Omron Sysmac Studio project NX1P2_e_NS_EmSimulação (Sysmac Studio 1.41.0.10, StandardProject)

# Controller new_Controller_0: NJ101-1020 version 1.12
Units and slaves: Power Supply : NJ-Px3001; CPU : NJ101-1020
Task PrimaryTask (priority 4, period or condition 2000): Programas

VAR_GLOBAL
    CH_Ciclo : BOOL;  (* published *)
    LMP_VM : BOOL;  (* published *)
    LMP_VD : BOOL;  (* published *)
    LMP_AM : BOOL;  (* published *)
    Chave1 : BOOL;  (* published *)
    Chave2 : BOOL;  (* published *)
    Memo_Produto1 : ARRAY[0..9] OF LREAL;  (* published *)
    Memo_Produção : ARRAY[0..9] OF LREAL;  (* published *)
    Memo_Produto2 : ARRAY[0..9] OF LREAL;  (* published *)
    TempoVM : TIME;  (* published *)
    TempoVD : TIME;  (* published *)
    TempoAM : TIME;  (* published *)
END_VAR

PROGRAM Programas
VAR
    TON_3 : TON;
    TON_1 : TON;
    TON_2 : TON;
    Ax_LMP_AM : BOOL;
END_VAR
VAR_EXTERNAL
    CH_Ciclo : BOOL;
    LMP_VM : BOOL;
    LMP_VD : BOOL;
    LMP_AM : BOOL;
    Chave1 : BOOL;
    Chave2 : BOOL;
    Memo_Produto1 : ARRAY[0..9] OF LREAL;
    Memo_Produção : ARRAY[0..9] OF LREAL;
    Memo_Produto2 : ARRAY[0..9] OF LREAL;
    TempoVM : TIME;
    TempoVD : TIME;
    TempoAM : TIME;
END_VAR
VAR
    _p1 : BOOL;
    _p2 : BOOL;
END_VAR

(* Section Semáforo: ladder, written here as Structured Text *)

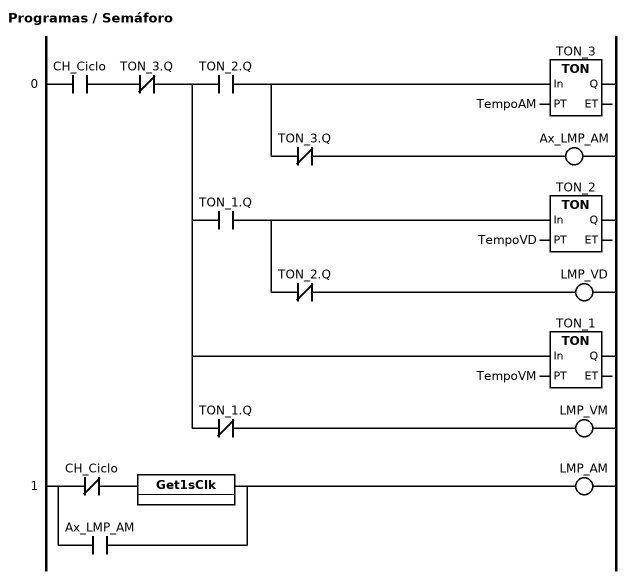
(* Rung 0 *)
_p1 := CH_Ciclo AND NOT TON_3.Q;
_p2 := CH_Ciclo AND NOT TON_3.Q AND TON_2.Q;
TON_3(In := _p2, PT := TempoAM);
Ax_LMP_AM := _p2 AND NOT TON_3.Q;
TON_2(In := _p1 AND TON_1.Q, PT := TempoVD);
LMP_VD := _p1 AND TON_1.Q AND NOT TON_2.Q;
TON_1(In := _p1, PT := TempoVM);
LMP_VM := _p1 AND NOT TON_1.Q;
(* Rung 1 *)
LMP_AM := (NOT CH_Ciclo AND Get1sClk()) OR Ax_LMP_AM;

(* Section Receita: ladder, written here as Structured Text *)

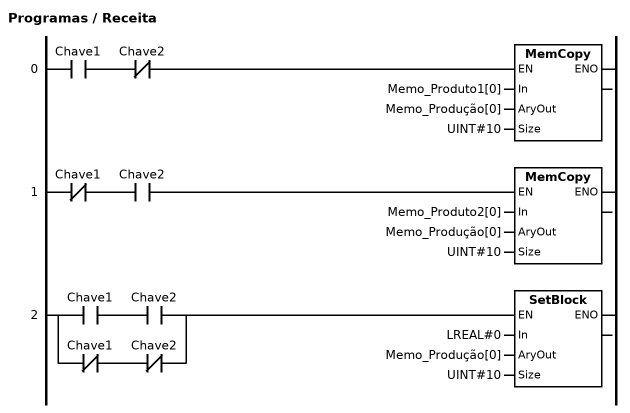
(* Rung 0 *)
IF Chave1 AND NOT Chave2 THEN
    MemCopy(In := Memo_Produto1[0], AryOut := Memo_Produção[0], Size := UINT#10);
END_IF;
(* Rung 1 *)
IF NOT Chave1 AND Chave2 THEN
    MemCopy(In := Memo_Produto2[0], AryOut := Memo_Produção[0], Size := UINT#10);
END_IF;
(* Rung 2 *)
IF (Chave1 AND Chave2) OR (NOT Chave1 AND NOT Chave2) THEN
    SetBlock(In := LREAL#0, AryOut := Memo_Produção[0], Size := UINT#10);
END_IF;
END_PROGRAM